ABB RobotStudio station: RobotStudio_20230302-170018.rsstn

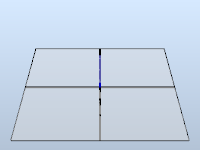
Station Station (saved by RobotStudio 22.1.9826.0)
Layout (positions relative to the parent item):
